{attribute 'qualified_only'}
{attribute 'strict'}
TYPE E_LaudaResponseError :
(
	NO_ERROR := 0,
	WRONG_ENTRY,
	WRONG_COMMAND,
	SYNTAX_ERROR,
	IMPERMISSABLE_VALUE,
	MODULE_OR_VALUE_NOT_AVAILABLE,
	ALL_SEGMENTS_IN_THE_PROGRAMMER_OCCUPIED,
	SETPOINT_NOT_POSSIBLE_WITH_ANALOG_SETPOINT_USED,
	EXTERNAL_TEMPERATURE_PROBE_MISSING,
	ANALOG_VALUE_NOT_PRESENT,
	SAFETY_MODE_CANT_START_IF_NOT_ENABLED,
	CANT_SET_VALUE_PROGRAMMER_RUNNING_OR_PAUSED,
	CANT_START_PROGRAMMER_ANALOG_SETPOINT_USED,
	CANT_ACTIVATE_FROM_SAFETY_MODE
);
END_TYPE

(* stored: Version 1.1.0.1, ProductVersion 3.1.4024.13
   DUT E_LaudaResponseError: Id {bc1c574f-42b3-0460-0ca9-4d087e2948ba} *)
